TYPE Wsl15_RegSegmentCfg :
STRUCT
	//fix byte inversion by defining them inverse...
	AnimationSync:BYTE;	
	BackgroundIntensity:eWsl15_Intensity;
	BackgroundColor:BYTE;
	SegmentMode:BYTE;

	//order in hw-config
	(*
	SegmentMode:BYTE;			
	BackgroundColor:BYTE;		
	BackgroundIntensity:eWsl15_Intensity;
	AnimationSync:BYTE;	
	*)
END_STRUCT
END_TYPE

(* stored: Version 1.1.0.1
   DUT Wsl15_RegSegmentCfg: Id {57e39055-4f4b-443c-9333-cd113dd7bde1} *)
